TYPE ST_ElementData :
(**************************************************************************************
 * 	Application		:	BoxControl Framework
 *	Revision		:	$Revision: 404529 $
 *	Revision date	:	$Date: 2018-04-23 08:21:38 +0200 (Mo., 23 Apr 2018) $
 *	Last changed by	:	$Author: b7bolm $
 *	URL				:	$URL: http://almscdc.swisslog.com/repo/SWPD/Development/BoxControlFramework/20_Release/trunk/01_Software/BCF/BCF/JumpStart/20_Product/10_App/13_Elements/10_Lib/10_Conv/01_DUTs/ST_ElementData.TcDUT $
 *
 *	Purpose			:	Element data - All data which are used internally. 
 *						External accessable over property (Read only)
 *
 * ------------------------------------------------------------------------------------
 *	Copyright Swisslog [IP AG], Switzerland. All rights reserved.
 * 
 * ------------------------------------------------------------------------------------
 *	
 * 	Revision History: 
 *
 * 	VERSION			DATE			INITIALS			DESCRIPTION
 *	0.1				01.01.2001		swl					Example
 *
 **************************************************************************************)
STRUCT
	Init					: BOOL; // Initialized
	InitRunning				: BOOL; // Init ongoing
	OperationState			: ST_PositionState; // Information about the state
	FunctionOrder			: ST_FunctionOrders; // Result of all functions
	MemberList				: ST_ElementMemberList; // List of objects which are linkt to this element
	ErrorData				: ST_ElementErrorStruct; // All error structures
	ControlRequest			: ST_ControlRequest; // Control request
END_STRUCT
END_TYPE

(* stored: Version 1.1.0.1, ProductVersion 3.1.4022.12
   DUT ST_ElementData: Id {d39b6fb1-009f-4d60-8d89-3e34c030b5a3} *)
